(* IEC 61131-3 sources: CODESYS-IO-Visualization/CODESYS-IO-Visualization.fbsproj/Subs/Clock/ClockParsing, 12 files *)

(* ---- GetClockLocal.prg.st ---- *)
PROGRAM GetClockLocal

VAR_INPUT
	TZ: STRING := 'MT';  (* Supports: ET, CT, MT, ET *);
	DisableDST: BOOL := FALSE;
END_VAR

(* ---- GetDateLeapYear.prg.st ---- *)
PROGRAM GetDateLeapYear

VAR_INPUT
	Clock: DATE;
END_VAR

VAR_OUTPUT
	value: BOOL;
END_VAR

(* ---- GetDateMonth.prg.st ---- *)
PROGRAM GetDateMonth

VAR_INPUT
	Clock: DATE;
END_VAR

VAR_OUTPUT
	value: INT;
END_VAR

VAR
	leap: BOOL;
END_VAR

GetDayOfYear(Clock := Clock, value => value);

GetDateLeapYear(Clock := Clock, value => leap);

IF value < 32 THEN
	value := 1;
ELSIF leap THEN
	value := (value * 53 + 1668) / 1623;
ELSE
	value := (value * 53 + 1700) / 1620;
END_IF;

(* ---- GetDateYear.prg.st ---- *)
PROGRAM GetDateYear

VAR_INPUT
	Clock: DATE;
END_VAR

VAR_OUTPUT
	value: INT;
END_VAR

value := DWORD_TO_INT((DATE_TO_DWORD(Clock) + 43200) / 31557600 + 1970);

(* ---- GetDayOfMonth.prg.st ---- *)
PROGRAM GetDayOfMonth

VAR_INPUT
	Clock: DATE;
END_VAR

VAR_OUTPUT
	value: INT;
END_VAR

VAR
	leap: BOOL;
	MonthDays : ARRAY[1..12] OF INT :=[ 0,31,59,90,120,151,181,212,243,273,304,334 ];
END_VAR

GetDayOfYear(Clock := Clock, value => value);
GetDateLeapYear(Clock := Clock, value => leap);
value := value - BOOL_TO_INT(leap);

IF value > MonthDays[9] THEN
	IF value > MonthDays[11] THEN
		IF value > MonthDays[12] THEN
			value := value - MonthDays[12];
		ELSE
			value := value - MonthDays[11];
		END_IF;
	ELSE
		IF value > MonthDays[10] THEN
			value := value - MonthDays[10];
		ELSE
			value := value - MonthDays[9];
		END_IF;
	END_IF;
ELSIF value > MonthDays[5] THEN
	IF value > MonthDays[7] THEN
		IF value > MonthDays[8] THEN
			value := value - MonthDays[8];
		ELSE
			value := value - MonthDays[7];
		END_IF;
	ELSE
		IF value > MonthDays[6] THEN
			value := value - MonthDays[6];
		ELSE
			value := value - MonthDays[5];
		END_IF;
	END_IF;
ELSIF value > MonthDays[3] THEN
	IF value > MonthDays[4] THEN
		value := value - MonthDays[4];
	ELSE
		value := value - MonthDays[3];
	END_IF;
ELSE
	value := value + BOOL_TO_INT(leap);
	IF value > MonthDays[2] THEN
		value := value - MonthDays[2];
	END_IF;
END_IF;

(* ---- GetDayOfWeek.prg.st ---- *)
PROGRAM GetDayOfWeek

VAR_INPUT
	Clock: DATE;
END_VAR

VAR_OUTPUT
	value: INT;
END_VAR

// Monday = 1 ... Sunday = 7

value := DWORD_TO_INT((DATE_TO_DWORD(Clock) / 86400 + 3) MOD 7) + 1;

(* ---- GetDayOfYear.prg.st ---- *)
PROGRAM GetDayOfYear

VAR_INPUT
	Clock: DATE;
END_VAR

VAR_OUTPUT
	value: INT;
END_VAR

value := UDINT_TO_INT((DATE_TO_UDINT(Clock) / UDINT#86400) MOD UDINT#1461);
IF value > 729 THEN
	IF value > 1095 THEN
		value := value - 1095;
	ELSE
		value := value - 729;
	END_IF;
ELSIF value > 364 THEN
	value := value - 364;
ELSE
	value := value + 1;
END_IF;

(* ---- GetDTHour.prg.st ---- *)
PROGRAM GetDTHour

VAR_INPUT
	Clock: DT;
END_VAR

VAR_OUTPUT
	value: INT;
END_VAR

value := DWORD_TO_INT((DT_TO_DWORD(Clock) MOD 86400) / 3600);

(* ---- GetDTIsDST.prg.st ---- *)
PROGRAM GetDTIsDST

VAR_INPUT
	Clock: DT;
END_VAR

VAR
	month: INT; (* the current month *)
	day: INT;   (* the current day *)
	hour: INT;  (* the current hour (0 - 23), using Local Standard Time *)
	dow: INT;   (* the day of the week (1 = Monday, 7 = Sunday) using Local Standard Time *)
	prevSunday: INT;
END_VAR

VAR_OUTPUT
	IsDST: BOOL;
END_VAR

(* DST ON, second Sunday in March, it must be between 3/8 and 3/14 inclusive *)
(* DST OFF, first Sunday in November, it must be between 11/1 and 11/7 inclusive *)

GetDateMonth(Clock := DT_TO_DATE(Clock), value => month);
GetDayOfMonth(Clock := DT_TO_DATE(Clock), value => day);
GetDTHour(Clock := Clock, value => hour);
GetDayOfWeek(Clock := DT_TO_DATE(Clock), value => dow);

IF (month < 3 OR month > 11) THEN
	IsDST := FALSE;
	RETURN;
END_IF;

IF (month > 3 AND month < 11) THEN
	IsDST := TRUE;
	RETURN;
END_IF;

IF ((month = 11 AND day > 7) OR (month = 3 AND day < 8)) THEN
	IsDST := FALSE;
	RETURN;
END_IF;

IF (month = 3 AND day > 14) THEN
	IsDST := TRUE;
	RETURN;
END_IF;

(* If we get to here, it is either March 8 - 14 or November 1 - 7 *)
prevSunday := day - dow;

IF (month = 3) THEN
	IF (dow = 7) THEN
		IsDST := (hour > 1);
		RETURN;
	END_IF;

	IsDST := (prevSunday > 7 AND prevSunday < 15);
	RETURN;
END_IF;

(* If we get here, it is November 1 - 7 *)
IF (dow = 7) THEN
	IsDST := (hour < 2);
	RETURN;
END_IF;

IsDST := prevSunday < 1;

(* ---- GetDTMinute.prg.st ---- *)
PROGRAM GetDTMinute

VAR_INPUT
	Clock: DT;
END_VAR

VAR_OUTPUT
	value: INT;
END_VAR

value := DWORD_TO_INT(DT_TO_DWORD(Clock) MOD 3600) / 60;

(* ---- GetDTSecond.prg.st ---- *)
PROGRAM GetDTSecond

VAR_INPUT
	Clock: DT;
END_VAR

VAR_OUTPUT
	value: INT;
END_VAR

value := DWORD_TO_INT(DT_TO_DWORD(Clock) MOD 60);

(* ---- GetIsDST_1.prg.st ---- *)
PROGRAM GetIsDST_1

VAR_INPUT
	month: INT; (* the current month *)
	day: INT;   (* the current day *)
	hour: INT;  (* the current hour (0 - 23), using Local Standard Time *)
	dow: INT;   (* the day of the week (1 = Monday, 7 = Sunday) using Local Standard Time *)
END_VAR

VAR
	prevSunday: INT;
END_VAR

VAR_OUTPUT
	IsDST: BOOL;
END_VAR

(* DST ON, second Sunday in March, it must be between 3/8 and 3/14 inclusive *)
(* DST OFF, first Sunday in November, it must be between 11/1 and 11/7 inclusive *)

IF (month < 3 OR month > 11) THEN
	IsDST := FALSE;
	RETURN;
END_IF;

IF (month > 3 AND month < 11) THEN
	IsDST := TRUE;
	RETURN;
END_IF;

IF ((month = 11 AND day > 7) OR (month = 3 AND day < 8)) THEN
	IsDST := FALSE;
	RETURN;
END_IF;

IF (month = 3 AND day > 14) THEN
	IsDST := TRUE;
	RETURN;
END_IF;

(* If we get to here, it is either March 8 - 14 or November 1 - 7 *)
prevSunday := day - dow;

IF (month = 3) THEN
	IF (dow = 7) THEN
		IsDST := (hour > 1);
		RETURN;
	END_IF;

	IsDST := (prevSunday > 7 AND prevSunday < 15);
	RETURN;
END_IF;

(* If we get here, it is November 1 - 7 *)
IF (dow = 7) THEN
	IsDST := (hour < 2);
	RETURN;
END_IF;

IsDST := prevSunday < 1;
